// TIA Portal V17 export
// export: Created 2024-09-02T12:50:29.4773803Z, ExportSetting WithDefaults, DisplayName Totally Integrated Automation Portal, DisplayVersion V17, DisplayName TIA Portal Openness, DisplayVersion V17, DisplayName TIA Portal Version Control Interface, DisplayVersion V17, DisplayName STEP 7 Professional, DisplayVersion V17, DisplayName STEP 7 Safety, DisplayVersion V17, DisplayName WinCC Professional, DisplayVersion V17
TYPE "e_MGB"
// stored: IsFailsafeCompliant false
   STRUCT
      TasterTürAnfordern : Bool;   // Busmodul - Taster Anforderung Tür öffnen / Bus module - Push-button Door open request
      "res0.1" : Bool;   // Busmodul - Reserve / Bus module - reserve
      "res0.2" : Bool;   // Busmodul - Reserve / Bus module - reserve
      "res0.3" : Bool;   // Busmodul - Reserve / Bus module - reserve
      "res0.4" : Bool;   // Busmodul - Reserve / Bus module - reserve
      TasterTürQuitttieren : Bool;   // Busmodul - Taster Schliessen / Quitttieren / Bus module - close acknowledge button
      "res0.6" : Bool;   // Busmodul - Reserve / Bus module - reserve
      "res0.7" : Bool;   // Busmodul - Reserve / Bus module - reserve
      "res1.0" : Bool;   // Busmodul - Reserve / Bus module - reserve
      "res1.1" : Bool;   // Busmodul - Reserve / Bus module - reserve
      "res1.2" : Bool;   // Busmodul - Reserve / Bus module - reserve
      "res1.3" : Bool;   // Busmodul - Reserve / Bus module - reserve
      "res1.4" : Bool;   // Busmodul - Reserve / Bus module - reserve
      "res1.5" : Bool;   // Busmodul - Reserve / Bus module - reserve
      "res1.6" : Bool;   // Busmodul - Reserve / Bus module - reserve
      "res1.7" : Bool;   // Busmodul - Reserve / Bus module - reserve
      "MeldekontaktNot-Halt" : Bool;   // Notausmodul - Meldekontakt Not-Halt / Emergency stop module - signal contact Emergency stop
      "res2.1" : Bool;   // Notausmodul - Reserve / Emergency stop module - reserve
      "res2.2" : Bool;   // Notausmodul - Reserve / Emergency stop module - reserve
      "res2.3" : Bool;   // Notausmodul - Reserve / Emergency stop module - reserve
      "res2.4" : Bool;   // Notausmodul - Reserve / Emergency stop module - reserve
      "res2.5" : Bool;   // Notausmodul - Reserve / Emergency stop module - reserve
      "res2.6" : Bool;   // Notausmodul - Reserve / Emergency stop module - reserve
      "res2.7" : Bool;   // Notausmodul - Reserve / Emergency stop module - reserve
      Türstellung : Bool;   // Zuhaltemodul - Türstellung / Blocking module - Door position
      Riegelstellung : Bool;   // Zuhaltemodul - Riegelstellung / Blocking module - bolt position
      Zuhaltung : Bool;   // Zuhaltemodul - Zuhaltung / Blocking module - Blocking device
      "res3.3" : Bool;   // Zuhaltemodul - Reserve / Blocking module - reserve
      "res3.4" : Bool;   // Zuhaltemodul - Reserve / Blocking module - reserve
      "res3.5" : Bool;   // Zuhaltemodul - Reserve / Blocking module - reserve
      SK : Bool;   // Zuhaltemodul - SK (T&R) / Blocking module - SK (T&R)
      ÜK : Bool;   // Zuhaltemodul - ÜK (T&R&Z) / Blocking module - ÜK (T&R&Z)
      Error_diag : Bool;   // Diagnose - Error / Diagnosis - Error
      ErrorMgb_diag : Bool;   // Diagnose - Error MGB / Diagnosis - Error MGB
      "res4.2" : Bool;   // Diagnose - Reserve / Diagnosis - Reserve
      "res4.3" : Bool;   // Diagnose - Reserve / Diagnosis - Reserve
      "res4.4" : Bool;   // Diagnose - Reserve / Diagnosis - Reserve
      "res4.5" : Bool;   // Diagnose - Reserve / Diagnosis - Reserve
      "res4.6" : Bool;   // Diagnose - Reserve / Diagnosis - Reserve
      "res4.7" : Bool;   // Diagnose - Reserve / Diagnosis - Reserve
   END_STRUCT;
END_TYPE
